(* IEC 61131-3 sources: OpenPLC_v3/runtime/integration_test, 9 files *)

(* ---- modbusslave_discreteinput_false.st ---- *)
PROGRAM program0
  VAR
    DiscreteInput AT %IX0.0 : BOOL;
  END_VAR

  DiscreteInput := FALSE;
END_PROGRAM

CONFIGURATION Config0

  RESOURCE Res0 ON PLC
    TASK task0(INTERVAL := T#20ms,PRIORITY := 0);
    PROGRAM instance0 WITH task0 : program0;
  END_RESOURCE
END_CONFIGURATION

(* ---- modbusslave_discreteinput_true.st ---- *)
PROGRAM program0
  VAR
    DiscreteInput AT %IX0.0 : BOOL;
  END_VAR

  DiscreteInput := TRUE;
END_PROGRAM

CONFIGURATION Config0

  RESOURCE Res0 ON PLC
    TASK task0(INTERVAL := T#20ms,PRIORITY := 0);
    PROGRAM instance0 WITH task0 : program0;
  END_RESOURCE
END_CONFIGURATION

(* ---- modbusslave_holdingregister_md.st ---- *)
PROGRAM program0
  VAR
    HoldingRegisterInt AT %MD0 : DINT;
  END_VAR

  HoldingRegisterInt := HoldingRegisterInt;
END_PROGRAM

CONFIGURATION Config0

  RESOURCE Res0 ON PLC
    TASK task0(INTERVAL := T#20ms,PRIORITY := 0);
    PROGRAM instance0 WITH task0 : program0;
  END_RESOURCE
END_CONFIGURATION

(* ---- modbusslave_holdingregister_ml.st ---- *)
PROGRAM program0
  VAR
    HoldingRegisterInt AT %ML0 : LINT;
  END_VAR

  HoldingRegisterInt := HoldingRegisterInt;
END_PROGRAM

CONFIGURATION Config0

  RESOURCE Res0 ON PLC
    TASK task0(INTERVAL := T#20ms,PRIORITY := 0);
    PROGRAM instance0 WITH task0 : program0;
  END_RESOURCE
END_CONFIGURATION

(* ---- modbusslave_holdingregister_mw.st ---- *)
PROGRAM program0
  VAR
    HoldingRegisterInt AT %MW0 : INT;
  END_VAR

  HoldingRegisterInt := HoldingRegisterInt;
END_PROGRAM

CONFIGURATION Config0

  RESOURCE Res0 ON PLC
    TASK task0(INTERVAL := T#20ms,PRIORITY := 0);
    PROGRAM instance0 WITH task0 : program0;
  END_RESOURCE
END_CONFIGURATION

(* ---- modbusslave_holdingregister_qw.st ---- *)
PROGRAM program0
  VAR
    HoldingRegisterInt AT %QW0 : INT;
  END_VAR

  HoldingRegisterInt := HoldingRegisterInt;
END_PROGRAM

CONFIGURATION Config0

  RESOURCE Res0 ON PLC
    TASK task0(INTERVAL := T#20ms,PRIORITY := 0);
    PROGRAM instance0 WITH task0 : program0;
  END_RESOURCE
END_CONFIGURATION

(* ---- modbusslave_multiplecoils.st ---- *)
PROGRAM program0
  VAR
    Coil0 AT %QX0.0 : BOOL;
    Coil1 AT %QX0.1 : BOOL;
    Coil2 AT %QX0.2 : BOOL;
  END_VAR

  Coil0 := Coil0;

END_PROGRAM

CONFIGURATION Config0

  RESOURCE Res0 ON PLC
    TASK task0(INTERVAL := T#20ms,PRIORITY := 0);
    PROGRAM instance0 WITH task0 : program0;
  END_RESOURCE
END_CONFIGURATION

(* ---- modbusslave_singlecoil.st ---- *)
PROGRAM program0
  VAR
    Coil AT %QX0.0 : BOOL;
  END_VAR

  Coil := Coil;
END_PROGRAM

CONFIGURATION Config0

  RESOURCE Res0 ON PLC
    TASK task0(INTERVAL := T#20ms,PRIORITY := 0);
    PROGRAM instance0 WITH task0 : program0;
  END_RESOURCE
END_CONFIGURATION

(* ---- socketserver.st ---- *)
PROGRAM prog0
  VAR
    var_in : BOOL;
    var_out : BOOL;
  END_VAR

  var_out := var_in;
END_PROGRAM

CONFIGURATION Config0

  RESOURCE Res0 ON PLC
    TASK Main(INTERVAL := T#50ms,PRIORITY := 0);
    PROGRAM Inst0 WITH Main : prog0;
  END_RESOURCE
END_CONFIGURATION
